//==================================================================================================
//								RJM Maszyny sp. z o.o.
//									13.05.2022
//	Klasa bazowa dla podzespołów maszyny 
// 	v1.0	|| TC v 3.1.4024.29		|| - pierwsza wersja
//==================================================================================================
FUNCTION_BLOCK FB_StanMaszyny_Baza IMPLEMENTS ITF_StanMaszyny
VAR_INPUT
END_VAR
VAR_OUTPUT
END_VAR
VAR

END_VAR

//==================================================================================================
//								RJM Maszyny sp. z o.o.
//									13.05.2022
//	Obsługa stanu ABORTED  
// 	v1.0	|| TC v 3.1.4024.29		|| - pierwsza wersja
//==================================================================================================
METHOD SM_Aborted : BOOL
VAR_INPUT
END_VAR
END_METHOD

//==================================================================================================
//								RJM Maszyny sp. z o.o.
//									13.05.2022
//	Obsługa stanu ABORTING
// 	v1.0	|| TC v 3.1.4024.29		|| - pierwsza wersja
//==================================================================================================
METHOD SM_Aborting : BOOL
VAR_INPUT
END_VAR
END_METHOD

//==================================================================================================
//								RJM Maszyny sp. z o.o.
//									13.05.2022
//	Obsługa stanu CLEARING  
// 	v1.0	|| TC v 3.1.4024.29		|| - pierwsza wersja
//==================================================================================================
METHOD SM_Clearing : BOOL
VAR_INPUT
END_VAR
END_METHOD

//==================================================================================================
//								RJM Maszyny sp. z o.o.
//									13.05.2022
//	Obsługa stanu COMPLETE  
// 	v1.0	|| TC v 3.1.4024.29		|| - pierwsza wersja
//==================================================================================================
METHOD SM_Complete : BOOL
VAR_INPUT
END_VAR
END_METHOD

//==================================================================================================
//								RJM Maszyny sp. z o.o.
//									13.05.2022
//	Obsługa stanu COMPLITING  
// 	v1.0	|| TC v 3.1.4024.29		|| - pierwsza wersja
//==================================================================================================
METHOD SM_Completing : BOOL
VAR_INPUT
END_VAR
END_METHOD

//==================================================================================================
//								RJM Maszyny sp. z o.o.
//									13.05.2022
//	Obsługa stanu EXECUTE  
// 	v1.0	|| TC v 3.1.4024.29		|| - pierwsza wersja
//==================================================================================================
METHOD SM_Execute : BOOL
VAR_INPUT
END_VAR
END_METHOD

//==================================================================================================
//								RJM Maszyny sp. z o.o.
//									13.05.2022
//	Obsługa stanu HELD  
// 	v1.0	|| TC v 3.1.4024.29		|| - pierwsza wersja
//==================================================================================================
METHOD SM_Held : BOOL
VAR_INPUT
END_VAR
END_METHOD

//==================================================================================================
//								RJM Maszyny sp. z o.o.
//									13.05.2022
//	Obsługa stanu HOLDING - wsztrymanie pracy przez maszyne  
// 	v1.0	|| TC v 3.1.4024.29		|| - pierwsza wersja
//==================================================================================================
METHOD SM_Holding : BOOL
VAR_INPUT
END_VAR
END_METHOD

//==================================================================================================
//								RJM Maszyny sp. z o.o.
//									13.05.2022
//	Obsługa stanu IDLE - maszyna gotowado pracy  
// 	v1.0	|| TC v 3.1.4024.29		|| - pierwsza wersja
//==================================================================================================
METHOD SM_Idle : BOOL
VAR_INPUT
END_VAR
END_METHOD

//==================================================================================================
//								RJM Maszyny sp. z o.o.
//									13.05.2022
//	Obsługa stanu RESETTING  
// 	v1.0	|| TC v 3.1.4024.29		|| - pierwsza wersja
//==================================================================================================
METHOD SM_Resetting : BOOL
VAR_INPUT
END_VAR
END_METHOD

//==================================================================================================
//								RJM Maszyny sp. z o.o.
//									13.05.2022
//	Obsługa stanu STARTING  
// 	v1.0	|| TC v 3.1.4024.29		|| - pierwsza wersja
//==================================================================================================
METHOD SM_Starting : BOOL
VAR_INPUT
END_VAR
END_METHOD

//==================================================================================================
//								RJM Maszyny sp. z o.o.
//									13.05.2022
//	Obsługa stanu STOPPED  
// 	v1.0	|| TC v 3.1.4024.29		|| - pierwsza wersja
//==================================================================================================
METHOD SM_Stopped : BOOL
VAR_INPUT
END_VAR
END_METHOD

//==================================================================================================
//								RJM Maszyny sp. z o.o.
//									13.05.2022
//	Obsługa stanu STOPPING  
// 	v1.0	|| TC v 3.1.4024.29		|| - pierwsza wersja
//==================================================================================================
METHOD SM_Stopping : BOOL
VAR_INPUT
END_VAR
END_METHOD

//==================================================================================================
//								RJM Maszyny sp. z o.o.
//									13.05.2022
//	Obsługa stanu SUSPENDED - praca wstrzymana prze operatora  
// 	v1.0	|| TC v 3.1.4024.29		|| - pierwsza wersja
//==================================================================================================
METHOD SM_Suspended : BOOL
VAR_INPUT
END_VAR
END_METHOD

//==================================================================================================
//								RJM Maszyny sp. z o.o.
//									13.05.2022
//	Obsługa stanu SUSPENDING  
// 	v1.0	|| TC v 3.1.4024.29		|| - pierwsza wersja
//==================================================================================================
METHOD SM_Suspending : BOOL
VAR_INPUT
END_VAR
END_METHOD

//==================================================================================================
//								RJM Maszyny sp. z o.o.
//									13.05.2022
//	Obsługa stanu UNHOLDING  
// 	v1.0	|| TC v 3.1.4024.29		|| - pierwsza wersja
//==================================================================================================
METHOD SM_Unholding : BOOL
VAR_INPUT
END_VAR
END_METHOD

//==================================================================================================
//								RJM Maszyny sp. z o.o.
//									13.05.2022
//	Obsługa stanu UNSUSPENDING  
// 	v1.0	|| TC v 3.1.4024.29		|| - pierwsza wersja
//==================================================================================================
METHOD SM_Unsuspending : BOOL
VAR_INPUT
END_VAR
END_METHOD

END_FUNCTION_BLOCK

(* stored: Version 1.1.0.1, ProductVersion 3.1.4024.11
   POU FB_StanMaszyny_Baza: Id {668edb3e-1ce7-42b0-b717-b15f849c6a2a}, SpecialFunc None
   Method SM_Aborted: Id {e443d503-570c-46fa-86f4-e34b9c97e579}
   Method SM_Aborting: Id {7db677b0-5297-4145-9142-386d9fd4463c}
   Method SM_Clearing: Id {4b0ac309-9913-4fc0-bea6-afa95234a24d}
   Method SM_Complete: Id {1d3f95c9-3963-4f15-8720-1585c1134433}
   Method SM_Completing: Id {6140f4b7-556f-4e1d-a07b-65939719b0c1}
   Method SM_Execute: Id {381ae8a5-7073-456c-ac0a-7f23c483d823}
   Method SM_Held: Id {b7be618f-33a5-47e3-a43b-f78a63ccf04b}
   Method SM_Holding: Id {6cc3c06b-3302-459f-a02b-e3a71306bbe7}
   Method SM_Idle: Id {b456fd2e-093f-4a2a-a9f1-2140b209cba7}
   Method SM_Resetting: Id {2e1500e4-ac96-4dab-a11e-ae0089d48561}
   Method SM_Starting: Id {98954e97-213a-468e-8239-a2280b56b654}
   Method SM_Stopped: Id {db28fd3c-1862-4eb4-b4ad-5627491b3932}
   Method SM_Stopping: Id {e33adf5d-6995-4414-8e1b-6dac7b299b65}
   Method SM_Suspended: Id {7a2d412b-b637-46bb-ac6a-1f5eb72735bb}
   Method SM_Suspending: Id {35fad57c-9956-4a16-8341-da5bae4b9509}
   Method SM_Unholding: Id {75910719-60f6-4c1e-94d1-4e40cc992a72}
   Method SM_Unsuspending: Id {4f15a5d8-3680-4775-9efd-bc000b95ffc3} *)
